DATA_BLOCK "Debug"
VAR
  Bypass : Array[0..100] of Bool;
  Squence : Array[0..100] of Bool;
END_VAR
BEGIN
END_DATA_BLOCK
